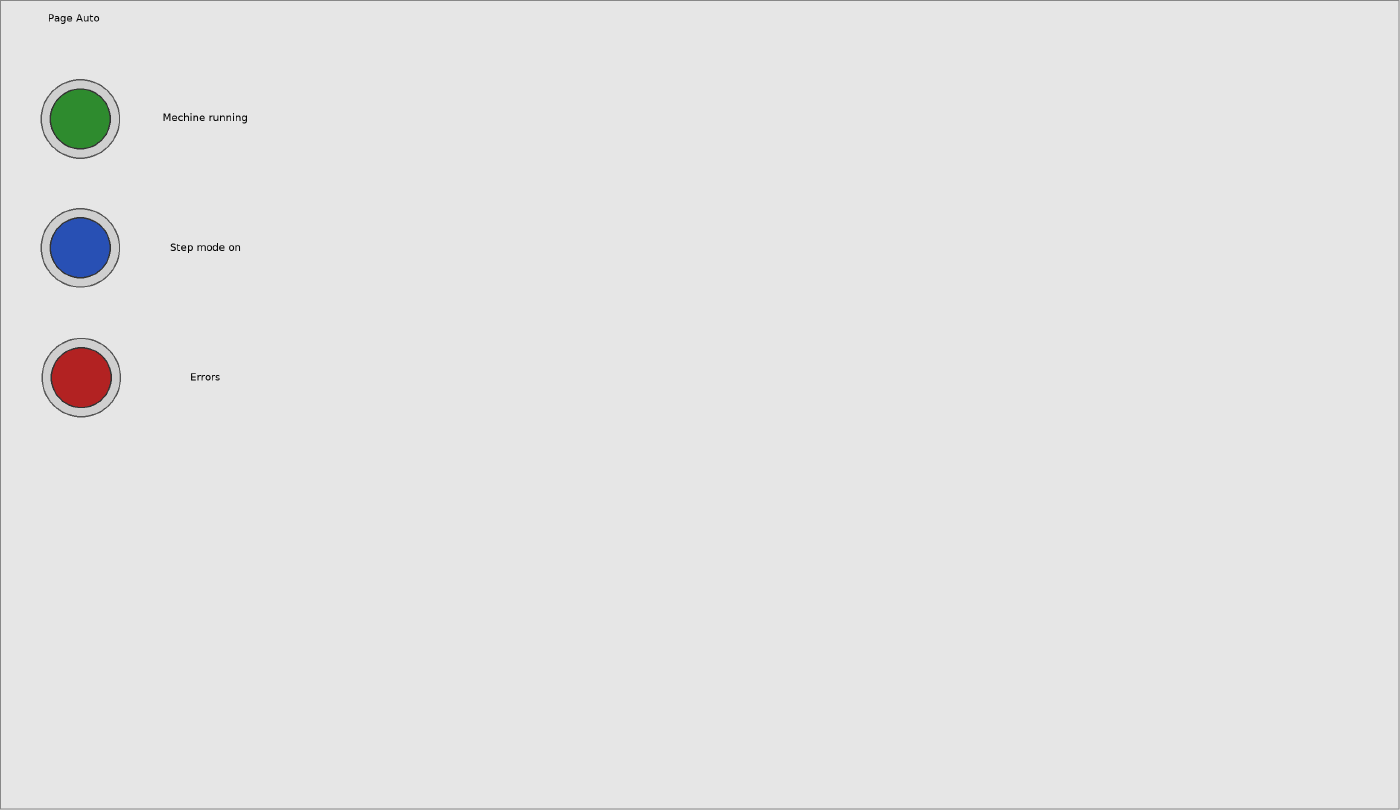
VISUALIZATION PageAuto  // 1520x880
    Label (5,5 150x30), "Page Auto"
    Label (148,113 150x30), "Mechine running"
    Label (148,254 150x30), "Step mode on"
    Lamp1 (37,79 100x100), variable: PRG_MachineControl.fbMachineControler.bRunning, style: Lamp-Lamp1-Green
    Lamp1 (37,219 100x100), variable: PRG_MachineControl.fbMachineControler.bStepMode, style: Lamp-Lamp1-Blue
    Lamp1 (38,360 100x100), variable: PRG_MachineControl.fbMachineControler.bError, style: Lamp-Lamp1-Red
    Label (148,395 150x30), "Errors"
END_VISUALIZATION

(* stored: Version 1.1.0.1, ProductVersion 3.1.4024.9
   Visu PageAuto: Id {be546244-d071-4731-a040-05c090ccddb8} *)
